TYPE OsCmd_MB_V1 :
   STRUCT
      Bon : Bool;   // Blocking on
      Boff : Bool;   // Blocking off
      Uon : Bool;   // Supression on
      Uoff : Bool;   // Supression off
      RX : Bool;   // Reset latched output
   END_STRUCT
END_TYPE

(* stored: Version 1.1.0.1, ProductVersion 3.1.4024.12
   DUT OsCmd_MB_V1: Id {572155cd-1cb7-4296-b8e0-698682541d76} *)
